# EPICS substitutions: evrSupport/Db/ioc/IOC-IN20-WS01pattern.substitutions
#
# Pattern records
file evrPatternAll.db {
#	    Device        ,  SLC Pattern Check LNK    , EVR/Trigger
#	                                                  Links
  pattern { DEVICE        ,        LINK4              , LINK5 , LINK6 , LINKD }
	  { IOC:IN20:WS01 ,         ""                ,  ""   ,  ""   ,  ""   }
}
file evrPatternProc.db {
  pattern { DEVICE }
	  { IOC:IN20:WS01}
}
